PROGRAM MAIN
VAR
END_VAR

END_PROGRAM

(* stored: Version 1.1.0.1
   POU MAIN: Id {cb89721e-a8c8-412a-96c3-f67b06e30055} *)
